INTERFACE I_TaskPool

METHOD PUBLIC FreeAllTasks
END_METHOD

METHOD PUBLIC GetTask : BOOL
VAR_OUTPUT
  result : I_CommandTask;
END_VAR
END_METHOD

END_INTERFACE

(* stored: Version 1.1.0.1
   Itf I_TaskPool: Id {20b53376-c05b-46c9-956c-bc2d71880f92}
   Method FreeAllTasks: Id {1420144b-8dd5-4774-aff1-c53a2528f5e1}
   Method GetTask: Id {7827d7f3-7258-4cb4-9452-9e70314da73b} *)
